PROGRAM PcTransmit
VAR
	fbPcTransmit_0 : fbPcTransmit;
	//fbLogTransmitMQTT : fbLogTransmitMQTT;
	isMqtt:BOOL;
END_VAR



IF isMqtt THEN
	//fbLogTransmitMQTT();
ELSE
	fbPcTransmit_0();
END_IF

END_PROGRAM

(* stored: Version 1.1.0.1, ProductVersion 3.1.4024.3
   POU PcTransmit: Id {fa84f91d-0024-00c8-17d0-8bb7ea7a8520}, SpecialFunc None *)
